{attribute addProperty BoxType "EJ3108-0000-0018"}
{attribute addProperty Id "AI_Standard_ChannelAT %I*ARRAY[0..7] OF AI_Standard_Channel_087F71C7256320WcStateAT %I*WcState_98A4DF7520.250InfoDataAT %I*InfoData_BC63D37F80100"}
{attribute addProperty CRC "864747523"}
{attribute addProperty SizeInBites "338"}
{attribute addProperty SizeInBytes "42.25"}
TYPE EJ3108_060F55FF :
STRUCT
	{attribute addProperty Name "AI_Standard_Channel"}
	AI_Standard_Channel : ARRAY[0..7] OF AI_Standard_Channel_087F71C7;
	{attribute addProperty Name "WcState"}
	WcState : WcState_98A4DF75;
	{attribute addProperty Name "InfoData"}
	InfoData : InfoData_BC63D37F;
END_STRUCT
END_TYPE

(* stored: Version 1.2.0.0, ProductVersion 3.1.4024.9
   DUT EJ3108_060F55FF: Id {91f5ea14-2f20-460c-b0ad-580aed80699f} *)
